TYPE READ_ADS_EVENT_HANDLEINFO :
STRUCT
	Enum			: DWORD;
	Count			: DWORD;
	
END_STRUCT
END_TYPE

(* stored: Version 1.1.0.1, ProductVersion 3.1.4024.12
   DUT READ_ADS_EVENT_HANDLEINFO: Id {1ba37464-4320-4354-b26e-595dd0fe5106} *)
